# EPICS StreamDevice protocol: imsApp/misc/report.proto
# Schneider Electric MDrivePlus Motor Protocol

InTerminator  = CR;
OutTerminator = CR LF;
ReplyTimeout  = 800;
ReadTimeout   = 100;
WriteTimeout  = 100;
ExtraInput    = Ignore;

# Reports from the controller
STATUS  { ReplyTimeout = 50; ReadTimeout = 10; InTerminator =; in "%.1/BOS([0-9,P=\-]*EOS)\r\n$/"; }

SAVING  { ReplyTimeout = 50; ReadTimeout = 10; InTerminator =; in "%.1/.*Want2([Save]*).*/"; }
SAVED_P { ReplyTimeout = 50; ReadTimeout = 10; InTerminator =; in "%.1/.*Saved ([0-9\-]*).*/"; }
